// SIMATIC STEP 7 (V5.x) project PLC_MST_WorkingClapans
// CPU: CPU 315-2 PN/DP
// station: P_ADR_BUS
// station: Hardware
// station: SIMATIC 300(2)(1)
// program: S7 Program(5)

SYMBOL_TABLE
"Arrays"	DB 1	DB 1
"Oscilation"	FB 1	FB 1
"S-Walce"	FB 2	FB 2
"GS Bottom&Top Sprusk"	FB 3	FB 3
"Hihgt Preassure Clapan"	FB 4	FB 4
"Service&Work"	FB 5	FB 5
"x0"	I 0.0	BOOL	// кн.Режим работы 1 пресс
"x1"	I 0.1	BOOL	// кн.Режим сервиса 1 пресс
"x2"	I 0.2	BOOL	// 1 Пресс прижать
"x3"	I 0.3	BOOL	// 1 пресс отжать
"x4"	I 0.4	BOOL	// кн.Режим работы 2 пресс работа
"x5"	I 0.5	BOOL	// кн.Режим работы 2 пресс сервис
"x6"	I 0.6	BOOL	// 2 Пресс прижать
"x7"	I 0.7	BOOL	// 2 пресс отжать
"x8"	I 1.0	BOOL	// Кн.Режм работы 3 пресс работа
"x9"	I 1.1	BOOL	// кн.Режим работы 3 пресс сервис
"x10"	I 1.2	BOOL	// 3 Пресс прижать
"x11"	I 1.3	BOOL	// 3 Пресс отжать
"x12"	I 1.4	BOOL	// кн.Осциляци выского давления сетка вкл
"x13"	I 1.5	BOOL	// кн.Осциляция высокого давления 1 пресс
"x14"	I 1.6	BOOL	// кн.Осциляция высокого давления 2 пресс вкл
"x15"	I 1.7	BOOL	// кн.Осциляция выского давления 3 пресс вкл
"x16"	I 2.0	BOOL	// кн.Клапан высокого давления сетка
"x17"	I 2.1	BOOL	// кн.Высокое давление 1 пресс
"x18"	I 2.2	BOOL	// кн. Включить Клапан высокого давления пресс 2
"x19"	I 2.3	BOOL	// кн.Клапан высокого давления 3 пресс
"x20"	I 2.4	BOOL	// кн.Осциляция орошения сукна 1 пресс
"x21"	I 2.5	BOOL	// кн.Осциляция орошения сукна 2 пресс
"x22"	I 2.6	BOOL	// Гидростанция прижима А
"x23"	I 2.7	BOOL	// Гидростанция прижима А пуск
"x24"	I 3.0	BOOL	// Гидростанция прижима В
"x25"	I 3.1	BOOL	// Гидростанция прижима В пуск
"x26"	I 3.2	BOOL	// кн.Гидростанция S-Walce A
"x27"	I 3.3	BOOL	// кн.Гидростанция S-Walce A пуск
"x28"	I 3.4	BOOL	// кн.Гидростанция S-Walce В
"x29"	I 3.5	BOOL	// кн.Гидростанция S-Walce В пуск
"x30"	I 3.6	BOOL	// кн.Вкл Гидростанция спрысков нижняя
"x31"	I 3.7	BOOL	// кн.Выкл Гидростанция спрысков нижняя
"x32"	I 4.0	BOOL	// кн.Вкл Нидростанция спрысков нижняя
"x33"	I 4.1	BOOL	// кн.Выкл Гидростанция спрысков верхняя
"x34"	I 4.2	BOOL	// кн.Стоп 1 пресс
"x35"	I 4.3	BOOL	// кн.Снять 1 пресс
"x36"	I 4.4	BOOL	// кн.Подвести 1 пресс
"x37"	I 4.5	BOOL	// кн.Прижим 1 пресс
"x38"	I 4.6	BOOL	// кн.Стоп 2 пресс
"x39"	I 4.7	BOOL	// кн.Снять 2 пресс
"x40"	I 5.0	BOOL	// кн.Подвести 2 пресс
"x41"	I 5.1	BOOL	// кн.Прижать 2 пресс
"x42"	I 5.2	BOOL	// Замок выкл
"x43"	I 5.3	BOOL	// Замок вкл
"x44"	I 5.4	BOOL	// кн.Стоп 3 пресс
"x45"	I 5.5	BOOL	// кн.Снять 3 пресс
"x46"	I 5.6	BOOL	// кн.Подвести 3 пресс
"x47"	I 5.7	BOOL	// кн.Прижать 3 пресс
"x48"	I 6.0	BOOL	// кн.Облегчть 3 пресс
"x49"	I 6.1	BOOL	// кн.Бомбировка 3 пресс выкл
"x50"	I 6.2	BOOL	// кн.Бомбировка 3 пресс вкл
"x51"	I 6.3	BOOL	// кн.Прижать сеткоповоротный вал
"x52"	I 6.4	BOOL	// кн.Прижим передающий вал 2
"x53"	I 6.5	BOOL	// кн.Прижать передающий вал 3 пресс
"x54"	I 6.6	BOOL	// Замок открыт
"x55"	I 6.7	BOOL	// Замок закрыт
"x56"	I 7.0	BOOL	// Замок открыт
"x57"	I 7.1	BOOL	// Замок закрыт
"x58"	I 7.2	BOOL
"x59"	I 7.3	BOOL
"x60"	I 7.4	BOOL
"x61"	I 7.5	BOOL
"x62"	I 7.6	BOOL
"x63"	I 7.7	BOOL
"x64"	I 8.0	BOOL
"x65"	I 8.1	BOOL
"x66"	I 8.2	BOOL
"x67"	I 8.3	BOOL
"x68"	I 8.4	BOOL
"x69"	I 8.5	BOOL
"x70"	I 8.6	BOOL
"x71"	I 8.7	BOOL
"x72"	I 9.0	BOOL
"x73"	I 9.1	BOOL
"x74"	I 9.2	BOOL
"x75"	I 9.3	BOOL
"x76"	I 9.4	BOOL
"x77"	I 9.5	BOOL
"x78"	I 9.6	BOOL
"x79"	I 9.7	BOOL
"x80"	I 10.0	BOOL
"x81"	I 10.1	BOOL
"x82"	I 10.2	BOOL
"x83"	I 10.3	BOOL
"x84"	I 10.4	BOOL
"x85"	I 10.5	BOOL
"x86"	I 10.6	BOOL
"x87"	I 10.7	BOOL
"x88"	I 11.0	BOOL
"x89"	I 11.1	BOOL
"x90"	I 11.2	BOOL
"x91"	I 11.3	BOOL
"x92"	I 11.4	BOOL
"x93"	I 11.5	BOOL
"x94"	I 11.6	BOOL
"x95"	I 11.7	BOOL
"x96"	I 12.0	BOOL
"x100"	I 12.1	BOOL
"x97"	I 12.2	BOOL
"x101"	I 12.3	BOOL
"x98"	I 12.4	BOOL
"x102"	I 12.5	BOOL
"x99"	I 12.6	BOOL
"x103"	I 12.7	BOOL
"x104"	I 13.0	BOOL
"x108"	I 13.1	BOOL
"x105"	I 13.2	BOOL
"x109"	I 13.3	BOOL
"x106"	I 13.4	BOOL
"x110"	I 13.5	BOOL
"x107"	I 13.6	BOOL
"x111"	I 13.7	BOOL
"x112"	I 14.0	BOOL
"x116"	I 14.1	BOOL
"x113"	I 14.2	BOOL
"x117"	I 14.3	BOOL
"x114"	I 14.4	BOOL
"x118"	I 14.5	BOOL
"x115"	I 14.6	BOOL
"x119"	I 14.7	BOOL
"x120"	I 15.0	BOOL
"x124"	I 15.1	BOOL
"x121"	I 15.2	BOOL
"x125"	I 15.3	BOOL
"x122"	I 15.4	BOOL
"x126"	I 15.5	BOOL
"x123"	I 15.6	BOOL
"x127"	I 15.7	BOOL
"x128"	I 16.0	BOOL
"x132"	I 16.1	BOOL
"x129"	I 16.2	BOOL
"x133"	I 16.3	BOOL
"x130"	I 16.4	BOOL
"x134"	I 16.5	BOOL
"x131"	I 16.6	BOOL
"x135"	I 16.7	BOOL
"x136"	I 17.0	BOOL
"x140"	I 17.1	BOOL
"x137"	I 17.2	BOOL
"x141"	I 17.3	BOOL
"x138"	I 17.4	BOOL
"x142"	I 17.5	BOOL
"x139"	I 17.6	BOOL
"x143"	I 17.7	BOOL
"x144"	I 18.0	BOOL
"x148"	I 18.1	BOOL
"x145"	I 18.2	BOOL
"x149"	I 18.3	BOOL
"x146"	I 18.4	BOOL
"x150"	I 18.5	BOOL
"x147"	I 18.6	BOOL
"x151"	I 18.7	BOOL
"x152"	I 19.0	BOOL
"x156"	I 19.1	BOOL
"x153"	I 19.2	BOOL
"x157"	I 19.3	BOOL
"x154"	I 19.4	BOOL
"x158"	I 19.5	BOOL
"x155"	I 19.6	BOOL
"x159"	I 19.7	BOOL
"x160"	I 20.0	BOOL
"x164"	I 20.1	BOOL
"x161"	I 20.2	BOOL
"x165"	I 20.3	BOOL
"x162"	I 20.4	BOOL
"x166"	I 20.5	BOOL
"x163"	I 20.6	BOOL
"x167"	I 20.7	BOOL
"x168"	I 21.0	BOOL
"x172"	I 21.1	BOOL
"x169"	I 21.2	BOOL
"x173"	I 21.3	BOOL
"x170"	I 21.4	BOOL
"x174"	I 21.5	BOOL
"x171"	I 21.6	BOOL
"x175"	I 21.7	BOOL
"x176"	I 22.0	BOOL
"x180"	I 22.1	BOOL
"x177"	I 22.2	BOOL
"x181"	I 22.3	BOOL
"x178"	I 22.4	BOOL
"x182"	I 22.5	BOOL
"x179"	I 22.6	BOOL
"x183"	I 22.7	BOOL
"x184"	I 23.0	BOOL
"x188"	I 23.1	BOOL
"x185"	I 23.2	BOOL
"x189"	I 23.3	BOOL
"x186"	I 23.4	BOOL
"x190"	I 23.5	BOOL
"x187"	I 23.6	BOOL
"x191"	I 23.7	BOOL
"x192"	I 24.0	BOOL
"x196"	I 24.1	BOOL
"x193"	I 24.2	BOOL
"x197"	I 24.3	BOOL
"x194"	I 24.4	BOOL
"x198"	I 24.5	BOOL
"x195"	I 24.6	BOOL
"x199"	I 24.7	BOOL
"x200"	I 25.0	BOOL
"x204"	I 25.1	BOOL
"x201"	I 25.2	BOOL
"x205"	I 25.3	BOOL
"x202"	I 25.4	BOOL
"x206"	I 25.5	BOOL
"x203"	I 25.6	BOOL
"x207"	I 25.7	BOOL
"x208"	I 26.0	BOOL
"x212"	I 26.1	BOOL
"x209"	I 26.2	BOOL
"x213"	I 26.3	BOOL
"x210"	I 26.4	BOOL
"x214"	I 26.5	BOOL
"x211"	I 26.6	BOOL
"x215"	I 26.7	BOOL
"x216"	I 27.0	BOOL
"x220"	I 27.1	BOOL
"x217"	I 27.2	BOOL
"x221"	I 27.3	BOOL
"x218"	I 27.4	BOOL
"x222"	I 27.5	BOOL
"x219"	I 27.6	BOOL
"x223"	I 27.7	BOOL
"x224"	I 28.0	BOOL
"x228"	I 28.1	BOOL
"x225"	I 28.2	BOOL
"x229"	I 28.3	BOOL
"x226"	I 28.4	BOOL
"x230"	I 28.5	BOOL
"x227"	I 28.6	BOOL	// Проток есть на 3 прессе
"x231"	I 28.7	BOOL
"x232"	I 29.0	BOOL
"x236"	I 29.1	BOOL	// Сигнал с ПРВ,сетка во вращении
"x233"	I 29.2	BOOL
"x237"	I 29.3	BOOL	// Сигнал с ПРВ,работа 3 приводов(1,2 пресс + пикап)
"x234"	I 29.4	BOOL
"x238"	I 29.5	BOOL	// Сигнал с ПРВ,3 пресс в работе
"x235"	I 29.6	BOOL
"x239"	I 29.7	BOOL	// Сигнал работы насос выского давления
"x240"	I 30.0	BOOL
"x244"	I 30.1	BOOL
"x241"	I 30.2	BOOL
"x245"	I 30.3	BOOL
"x242"	I 30.4	BOOL
"x246"	I 30.5	BOOL
"x243"	I 30.6	BOOL
"x247"	I 30.7	BOOL
"x248"	I 31.0	BOOL
"x252"	I 31.1	BOOL
"x249"	I 31.2	BOOL
"x253"	I 31.3	BOOL	// Дискретный датчик температуры ГС 1+3
"x250"	I 31.4	BOOL
"x254"	I 31.5	BOOL	// Дискретный датчик уровня масла ГС 1+3
"x251"	I 31.6	BOOL
"x255"	I 31.7	BOOL
"Delay_2tim"	MW 2	WORD	// Время задержки с панели на включение пресса
"CYCL_EXC"	OB 1	OB 1	// Cycle Execution
"Prog2"	OB 2	OB 2	// S-Walce
"Prog3"	OB 3	OB 3	// Sprusk
"y0"	Q 0.0	BOOL	// Лампа 1 пресс в режиме работы
"y1"	Q 0.1	BOOL	// Лампа пресс 1 в режиме сервис
"y2"	Q 0.2	BOOL	// Лампа 1 пресс прижать
"y3"	Q 0.3	BOOL	// Лампа 1 пресс отжать
"y4"	Q 0.4	BOOL	// Лампа 2 пресс в режиме работы
"y5"	Q 0.5	BOOL	// Лампа 2 пресс в режиме сервиса
"y6"	Q 0.6	BOOL	// Лампа 2 пресс прижать
"y7"	Q 0.7	BOOL	// Лампа 2 пресс отжать
"y8"	Q 1.0	BOOL	// Лампа 3 пресс в режиме работы
"y9"	Q 1.1	BOOL	// Лампа 3 пресс в режиме сервиса
"y10"	Q 1.2	BOOL	// Лампа 3 пресс прижать
"y11"	Q 1.3	BOOL	// Лампа 3 пресс отжать
"y12"	Q 1.4	BOOL	// Лампа выключена осциляция высокого давления сетки
"y13"	Q 1.5	BOOL	// Лампа включена рсциляция высокго давления сетка
"y14"	Q 1.6	BOOL	// Лампа выключена осциляция выского давления 1 пресс
"y15"	Q 1.7	BOOL	// Лампа включена Осциляция выского давления 1 пресс
"y16"	Q 2.0	BOOL	// Лампа выключена осциляция выского давления 2 пресс
"y17"	Q 2.1	BOOL	// Лампа включена осциляция выского давления 2 пресс
"y18"	Q 2.2	BOOL	// Лампа выключена осциляция высокого давления 3 пресс
"y19"	Q 2.3	BOOL	// Лампа включена осциляция высокого давления 3 пресс
"y20"	Q 2.4	BOOL	// Лампа выключен клапан высокого давления сетка
"y21"	Q 2.5	BOOL	// Лампа включен клапан высокого давления сетка
"y22"	Q 2.6	BOOL	// Лампа выключен клапан высокого давления пресс 1
"y23"	Q 2.7	BOOL	// Лампа включен Клапан высокого давления 1 пресс
"y24"	Q 3.0	BOOL	// Лампа выключен клапан высокого давления пресс 2
"y25"	Q 3.1	BOOL	// Лампа включен клапан высокого давления пресс 2
"y26"	Q 3.2	BOOL	// Лампа выключен клапан высокого давления пресс 3
"y27"	Q 3.3	BOOL	// Лампа включен клапан высокого давления пресс 3
"y28"	Q 3.4	BOOL	// Лампа выключена осциляция орошающего спрыска 1 пресс
"y29"	Q 3.5	BOOL	// Лампа включена осциляция орошающего спрыска 1 пресс
"y30"	Q 3.6	BOOL	// Лампа выключена осциляция орошающего спрыска 1 пресс
"y31"	Q 3.7	BOOL	// Лампа включена осциляция орошающего спрыска 2 пресс
"y32"	Q 4.0	BOOL	// Лампа вкл прижим А
"y33"	Q 4.1	BOOL	// Лампа выкл. Гидростанция прижима А&B
"y34"	Q 4.2	BOOL	// Лампа вкл прижим В
"y35"	Q 4.3	BOOL	// Лампа работы гидростанция S-Walke A
"y36"	Q 4.4	BOOL	// Лампа отключен. S-Walke A&B
"y37"	Q 4.5	BOOL	// Лампа работы гидростанция S-Walke B
"y38"	Q 4.6	BOOL	// Лампа выключена ГС спрысков нижняя
"y39"	Q 4.7	BOOL	// Лампа включена ГС спрысков нижняя
"y40"	Q 5.0	BOOL	// Лампа выключена ГС спрысков верхняя
"y41"	Q 5.1	BOOL	// Лампа включена ГС спрысков верхняя
"y42"	Q 5.2	BOOL	// Лампа Стоп 1й прес
"y43"	Q 5.3	BOOL	// Лампа зняти 1й прес
"y44"	Q 5.4	BOOL	// Лампа подвод 1й прес
"y45"	Q 5.5	BOOL	// Лампа прижать 1й прес
"y46"	Q 5.6	BOOL	// Лампа стоп 2й прес
"y47"	Q 5.7	BOOL	// Лампа зняти 2й прес
"y48"	Q 6.0	BOOL	// Лампа подвод 2й прес
"y49"	Q 6.1	BOOL	// Лампа прижати 2й прес
"y50"	Q 6.2	BOOL	// Лампа замок выкл
"y51"	Q 6.3	BOOL	// Лампа замок вкл
"y52"	Q 6.4	BOOL	// Лампа останов 3й прес
"y53"	Q 6.5	BOOL	// Лампа зняти 3й прес
"y54"	Q 6.6	BOOL	// Замок открыт
"y55"	Q 6.7	BOOL	// Лампа прижати 3й прес
"y56"	Q 7.0	BOOL	// Замок открыт
"y57"	Q 7.1	BOOL	// Лампа выключена бомбировка 3 пресс
"y58"	Q 7.2	BOOL	// Лампа включена бомбировка 3 пресс
"y59"	Q 7.3	BOOL	// Бомбировка вкл пресс 3
"y60"	Q 7.4	BOOL	// Клапан замка 1
"y61"	Q 7.5	BOOL	// Клапан замка 2
"y62"	Q 7.6	BOOL
"y63"	Q 7.7	BOOL
"y64"	Q 8.0	BOOL
"y65"	Q 8.1	BOOL
"y66"	Q 8.2	BOOL
"y67"	Q 8.3	BOOL
"y68"	Q 8.4	BOOL
"y69"	Q 8.5	BOOL
"y70"	Q 8.6	BOOL
"y71"	Q 8.7	BOOL
"y72"	Q 9.0	BOOL
"y73"	Q 9.1	BOOL
"y74"	Q 9.2	BOOL
"y75"	Q 9.3	BOOL
"y76"	Q 9.4	BOOL
"y77"	Q 9.5	BOOL
"y78"	Q 9.6	BOOL
"y79"	Q 9.7	BOOL
"y80"	Q 10.0	BOOL
"y81"	Q 10.1	BOOL
"y82"	Q 10.2	BOOL
"y83"	Q 10.3	BOOL
"y84"	Q 10.4	BOOL
"y85"	Q 10.5	BOOL
"y86"	Q 10.6	BOOL
"y87"	Q 10.7	BOOL
"y88"	Q 11.0	BOOL
"y89"	Q 11.1	BOOL
"y90"	Q 11.2	BOOL
"y91"	Q 11.3	BOOL
"y92"	Q 11.4	BOOL
"y93"	Q 11.5	BOOL
"y94"	Q 11.6	BOOL
"y95"	Q 11.7	BOOL
"y96"	Q 12.0	BOOL
"y100"	Q 12.1	BOOL
"y97"	Q 12.2	BOOL
"y101"	Q 12.3	BOOL
"y98"	Q 12.4	BOOL
"y102"	Q 12.5	BOOL
"y99"	Q 12.6	BOOL
"y103"	Q 12.7	BOOL	// Гидростанция S-Walce A
"y104"	Q 13.0	BOOL	// Гидростанция S-Walce В
"y108"	Q 13.1	BOOL
"y105"	Q 13.2	BOOL
"y109"	Q 13.3	BOOL
"y106"	Q 13.4	BOOL
"y110"	Q 13.5	BOOL
"y107"	Q 13.6	BOOL
"y111"	Q 13.7	BOOL	// Гидростанция спрысков верхняя
"y112"	Q 14.0	BOOL	// Гидростанция прижима А
"y116"	Q 14.1	BOOL
"y113"	Q 14.2	BOOL	// Гидростанция спырсков нижняя
"y117"	Q 14.3	BOOL
"y114"	Q 14.4	BOOL	// Гидростанция прижима В
"y118"	Q 14.5	BOOL
"y115"	Q 14.6	BOOL
"y119"	Q 14.7	BOOL
"y120"	Q 15.0	BOOL
"y124"	Q 15.1	BOOL	// Клапан ГС спрысков верхний
"y121"	Q 15.2	BOOL
"y125"	Q 15.3	BOOL
"y122"	Q 15.4	BOOL
"y126"	Q 15.5	BOOL	// Клапан высокого давления пресс 1
"y123"	Q 15.6	BOOL
"y127"	Q 15.7	BOOL	// Клапан высокго давления пресс 2
"y128"	Q 16.0	BOOL	// Клапан высокого давления пресс 3
"y132"	Q 16.1	BOOL
"y129"	Q 16.2	BOOL	// Клапан высокого давления сетка
"y133"	Q 16.3	BOOL	// WE3 2 PRESS
"y130"	Q 16.4	BOOL	// Сигнал на ПРВ, Дозвіл работы 1,2 пресса+пикап
"y134"	Q 16.5	BOOL	// WE2 2 PRESS
"y131"	Q 16.6	BOOL	// Сигнал на ПРВ,Запрет включения 3 пресса
"y135"	Q 16.7	BOOL	// WE1.1 2 PRESS
"y136"	Q 17.0	BOOL	// WE 1.2 2PRESS
"y140"	Q 17.1	BOOL
"y137"	Q 17.2	BOOL	// 2 пресс отжать
"y141"	Q 17.3	BOOL	// Прижим передающий вал 2 пресс
"y138"	Q 17.4	BOOL	// 2 пресс прижать
"y142"	Q 17.5	BOOL	// Отжать передающий вал 3 пресс
"y139"	Q 17.6	BOOL
"y143"	Q 17.7	BOOL	// Прижать передающий вал 3 пресс
"y144"	Q 18.0	BOOL	// Прижать сеткоповоротный вал
"y148"	Q 18.1	BOOL	// WE5.1 3 PRESS
"y145"	Q 18.2	BOOL	// WE3 1 PRESS
"y149"	Q 18.3	BOOL	// WE5.2 3 PRESS
"y146"	Q 18.4	BOOL	// WE2.1 1 PRESS
"y150"	Q 18.5	BOOL	// WE4.1 3 PRESS
"y147"	Q 18.6	BOOL	// WE2.2 1 PRESS
"y151"	Q 18.7	BOOL	// WE 4.2 3 PRESS
"y152"	Q 19.0	BOOL	// WE6 3 PRESS
"y156"	Q 19.1	BOOL	// 1 пресс прижать
"y153"	Q 19.2	BOOL	// 1 пресс прижать WE4
"y157"	Q 19.3	BOOL	// 1 пресс отжать WE4
"y154"	Q 19.4	BOOL	// 1 пресс прижать WE4 A
"y158"	Q 19.5	BOOL
"y155"	Q 19.6	BOOL	// 1 пресс отжать WE4 A
"y159"	Q 19.7	BOOL
"y160"	Q 20.0	BOOL	// 3 пресс прижать
"y164"	Q 20.1	BOOL	// Клапан осциляции выского давления 1 пресс
"y161"	Q 20.2	BOOL	// 3 пресс отжать
"y165"	Q 20.3	BOOL
"y162"	Q 20.4	BOOL	// Клапан осциляции высокого давления сетки
"y166"	Q 20.5	BOOL	// Клапан осциляции выского давления 2 пресс
"y163"	Q 20.6	BOOL	// Клапан осциляции выского давления 3 пресс
"y167"	Q 20.7	BOOL
"t0"	T 0	TIMER	// Таймер прерывания 1с
"t1"	T 1	TIMER	// Таймер прерывания 1с
"t2"	T 2	TIMER	// Задержка на разрешение включения пресса
"t3"	T 3	TIMER	// Задержка на разрешение включения пресса
"VAT_1"	VAT 1	
END_SYMBOL_TABLE

FUNCTION_BLOCK "Oscilation"	// FB 1
VERSION : 0.1
VAR_TEMP
  DatArray : ARRAY  [0 .. 5 ] OF INT ;
END_VAR
BEGIN
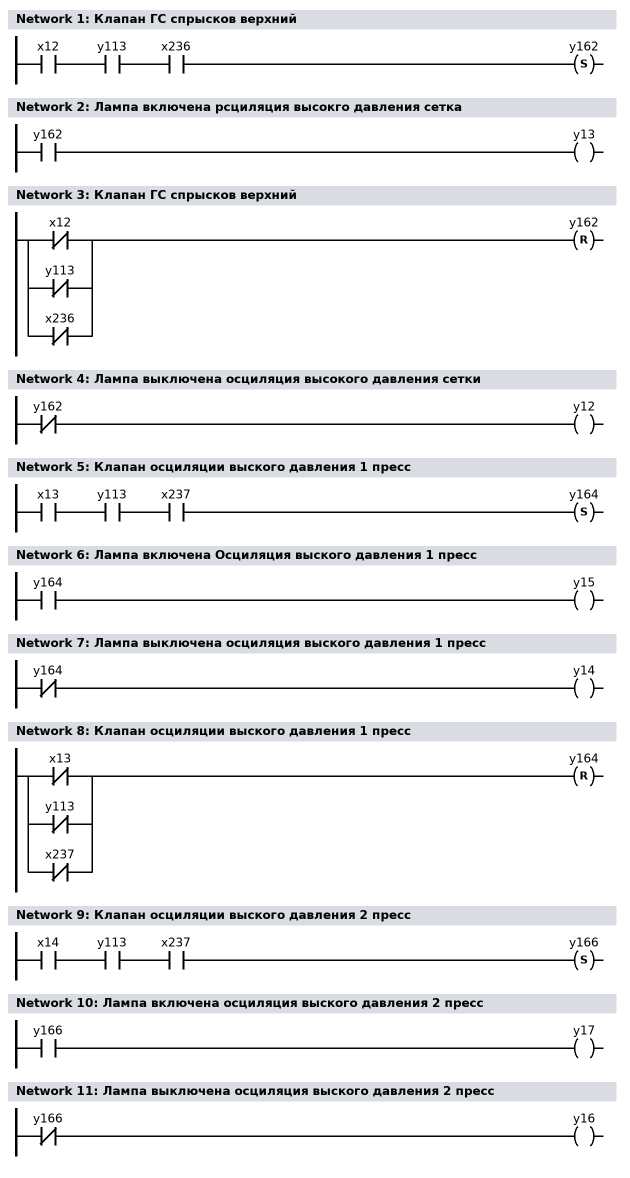
NETWORK
TITLE = Клапан ГС спрысков верхний
      A     "x12";
      A     "y113";
      A     "x236";
      S     "y162";
NETWORK
TITLE = Лампа включена рсциляция высокго давления сетка
      A     "y162";
      =     "y13";
NETWORK
TITLE = Клапан ГС спрысков верхний
      ON    "x12";
      ON    "y113";
      ON    "x236";
      R     "y162";
NETWORK
TITLE = Лампа выключена осциляция высокого давления сетки
      AN    "y162";
      =     "y12";
NETWORK
TITLE = Клапан осциляции выского давления 1 пресс
      A     "x13";
      A     "y113";
      A     "x237";
      S     "y164";
NETWORK
TITLE = Лампа включена Осциляция выского давления 1 пресс
      A     "y164";
      =     "y15";
NETWORK
TITLE = Лампа выключена осциляция выского давления 1 пресс
      AN    "y164";
      =     "y14";
NETWORK
TITLE = Клапан осциляции выского давления 1 пресс
      ON    "x13";
      ON    "y113";
      ON    "x237";
      R     "y164";
NETWORK
TITLE = Клапан осциляции выского давления 2 пресс
      A     "x14";
      A     "y113";
      A     "x237";
      S     "y166";
NETWORK
TITLE = Лампа включена осциляция выского давления 2 пресс
      A     "y166";
      =     "y17";
NETWORK
TITLE = Лампа выключена осциляция выского давления 2 пресс
      AN    "y166";
      =     "y16";
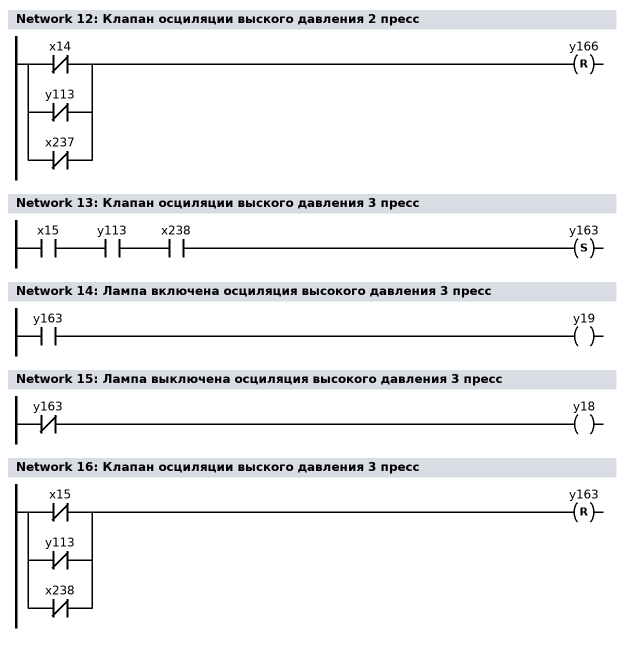
NETWORK
TITLE = Клапан осциляции выского давления 2 пресс
      ON    "x14";
      ON    "y113";
      ON    "x237";
      R     "y166";
NETWORK
TITLE = Клапан осциляции выского давления 3 пресс
      A     "x15";
      A     "y113";
      A     "x238";
      S     "y163";
NETWORK
TITLE = Лампа включена осциляция высокого давления 3 пресс
      A     "y163";
      =     "y19";
NETWORK
TITLE = Лампа выключена осциляция высокого давления 3 пресс
      AN    "y163";
      =     "y18";
NETWORK
TITLE = Клапан осциляции выского давления 3 пресс
      ON    "x15";
      ON    "y113";
      ON    "x238";
      R     "y163";
END_FUNCTION_BLOCK

FUNCTION_BLOCK "S-Walce"	// FB 2
VERSION : 0.1
BEGIN
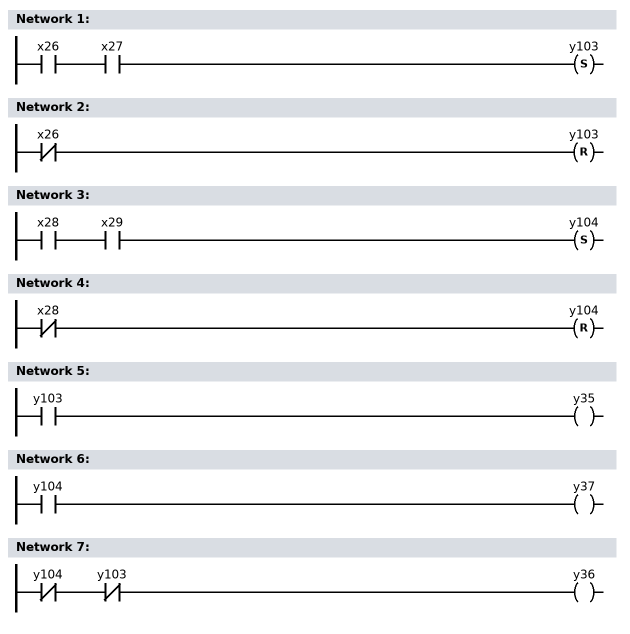
NETWORK
TITLE =
      A     "x26";
      A     "x27";
      S     "y103";
NETWORK
TITLE =
      AN    "x26";
      R     "y103";
NETWORK
TITLE =
      A     "x28";
      A     "x29";
      S     "y104";
NETWORK
TITLE =
      AN    "x28";
      R     "y104";
NETWORK
TITLE =
      A     "y103";
      =     "y35";
NETWORK
TITLE =
      A     "y104";
      =     "y37";
NETWORK
TITLE =
      AN    "y104";
      AN    "y103";
      =     "y36";
END_FUNCTION_BLOCK

FUNCTION_BLOCK "GS Bottom&Top Sprusk"	// FB 3
VERSION : 0.1
VAR_TEMP
  m0 : BOOL ;	//Аварийный сигнал с ГС 1+3
END_VAR
BEGIN
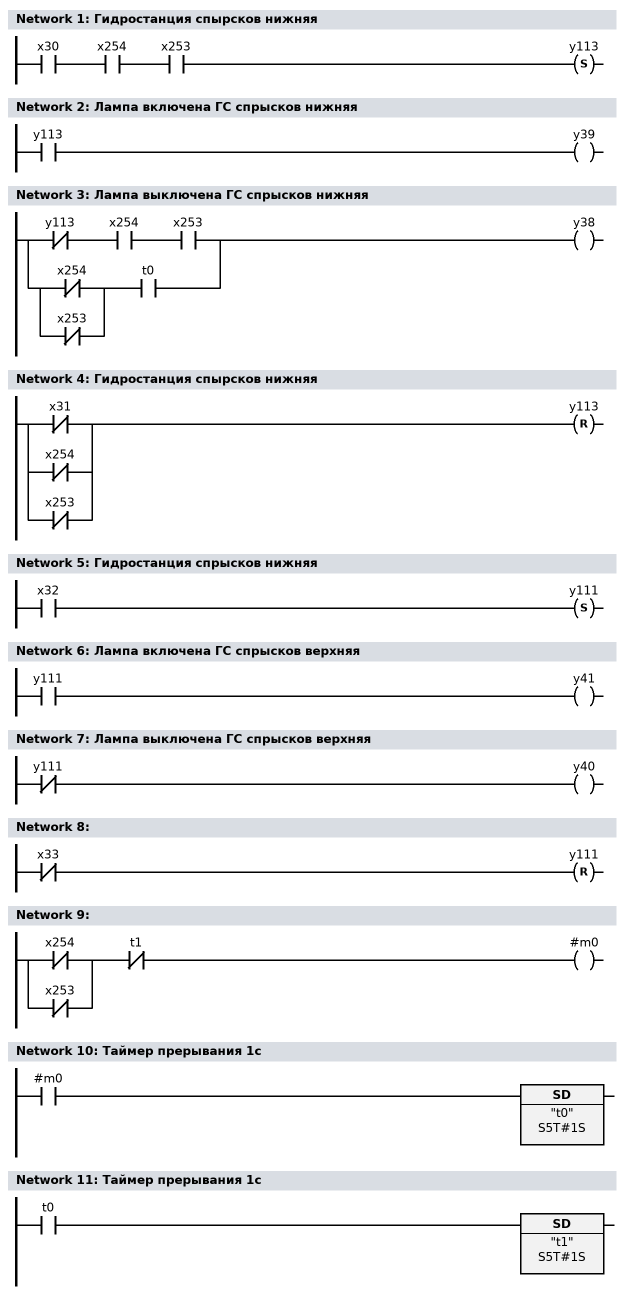
NETWORK
TITLE = Гидростанция спырсков нижняя
      A     "x30";
      A     "x254";
      A     "x253";
      S     "y113";
NETWORK
TITLE = Лампа включена ГС спрысков нижняя
      A     "y113";
      =     "y39";
NETWORK
TITLE = Лампа выключена ГС спрысков нижняя
      AN    "y113";
      A     "x254";
      A     "x253";
      O;
      A(;
      ON    "x254";
      ON    "x253";
      );
      A     "t0";
      =     "y38";
NETWORK
TITLE = Гидростанция спырсков нижняя
      ON    "x31";
      ON    "x254";
      ON    "x253";
      R     "y113";
NETWORK
TITLE = Гидростанция спрысков нижняя
      A     "x32";
      S     "y111";
NETWORK
TITLE = Лампа включена ГС спрысков верхняя
      A     "y111";
      =     "y41";
NETWORK
TITLE = Лампа выключена ГС спрысков верхняя
      AN    "y111";
      =     "y40";
NETWORK
TITLE =
      AN    "x33";
      R     "y111";
NETWORK
TITLE =
//<force open>
      A(;
      ON    "x254";
      ON    "x253";
      );
      AN    "t1";
      =     #m0;
NETWORK
TITLE = Таймер прерывания 1с
      A     #m0;
      L     S5T#1S;
      SD    "t0";
NETWORK
TITLE = Таймер прерывания 1с
      A     "t0";
      L     S5T#1S;
      SD    "t1";
END_FUNCTION_BLOCK

FUNCTION_BLOCK "Hihgt Preassure Clapan"	// FB 4
TITLE = Hight Pressure Klapan
VERSION : 0.1
BEGIN
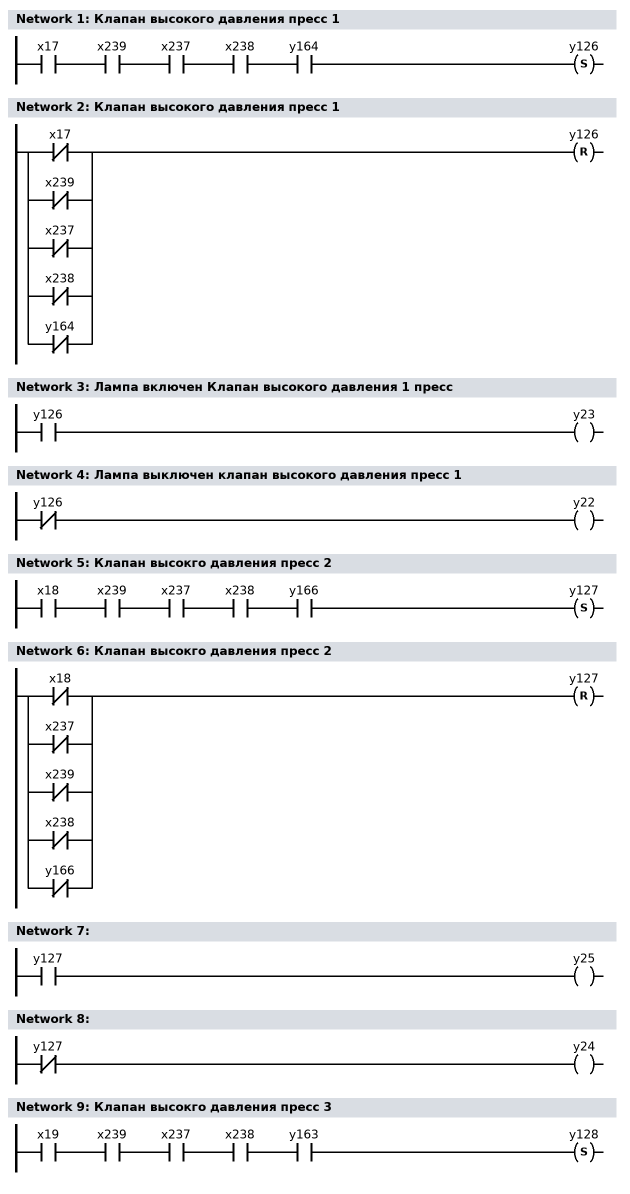
NETWORK
TITLE = Клапан высокого давления пресс 1
      A     "x17";
      A     "x239";
      A     "x237";
      A     "x238";
      A     "y164";
      S     "y126";
NETWORK
TITLE = Клапан высокого давления пресс 1
      ON    "x17";
      ON    "x239";
      ON    "x237";
      ON    "x238";
      ON    "y164";
      R     "y126";
NETWORK
TITLE = Лампа включен Клапан высокого давления 1 пресс
      A     "y126";
      =     "y23";
NETWORK
TITLE = Лампа выключен клапан высокого давления пресс 1
      AN    "y126";
      =     "y22";
NETWORK
TITLE = Клапан высокго давления пресс 2
      A     "x18";
      A     "x239";
      A     "x237";
      A     "x238";
      A     "y166";
      S     "y127";
NETWORK
TITLE = Клапан высокго давления пресс 2
      ON    "x18";
      ON    "x237";
      ON    "x239";
      ON    "x238";
      ON    "y166";
      R     "y127";
NETWORK
TITLE =
      A     "y127";
      =     "y25";
NETWORK
TITLE =
      AN    "y127";
      =     "y24";
NETWORK
TITLE = Клапан высокго давления пресс 3
      A     "x19";
      A     "x239";
      A     "x237";
      A     "x238";
      A     "y163";
      S     "y128";
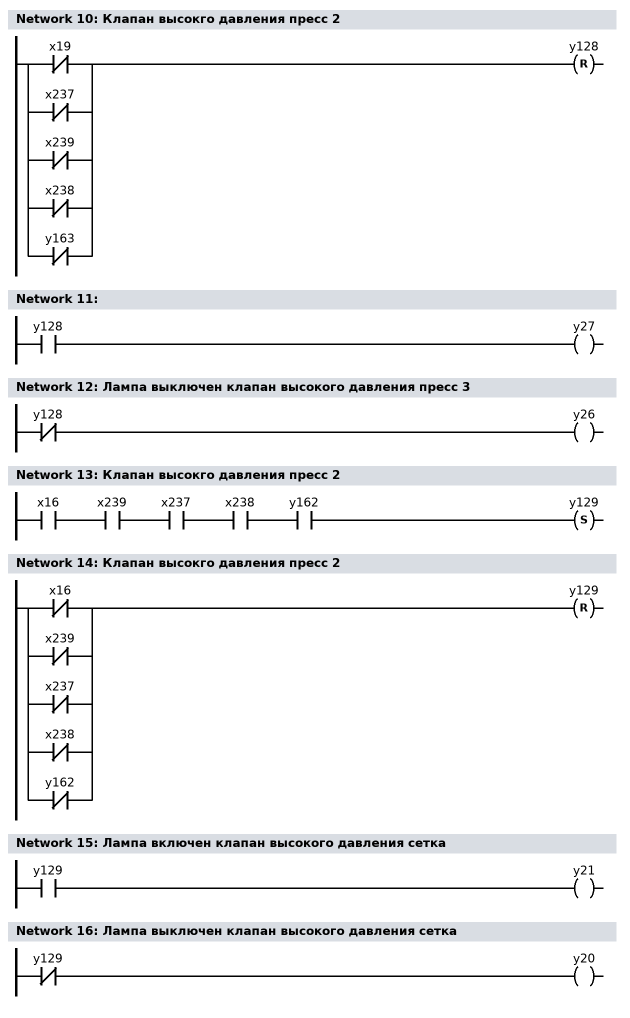
NETWORK
TITLE = Клапан высокго давления пресс 2
      ON    "x19";
      ON    "x237";
      ON    "x239";
      ON    "x238";
      ON    "y163";
      R     "y128";
NETWORK
TITLE =
      A     "y128";
      =     "y27";
NETWORK
TITLE = Лампа выключен клапан высокого давления пресс 3
      AN    "y128";
      =     "y26";
NETWORK
TITLE = Клапан высокго давления пресс 2
      A     "x16";
      A     "x239";
      A     "x237";
      A     "x238";
      A     "y162";
      S     "y129";
NETWORK
TITLE = Клапан высокго давления пресс 2
      ON    "x16";
      ON    "x239";
      ON    "x237";
      ON    "x238";
      ON    "y162";
      R     "y129";
NETWORK
TITLE = Лампа включен клапан высокого давления сетка
      A     "y129";
      =     "y21";
NETWORK
TITLE = Лампа выключен клапан высокого давления сетка
      AN    "y129";
      =     "y20";
END_FUNCTION_BLOCK

FUNCTION_BLOCK "Service&Work"	// FB 5
//SELECT MODE
//
VERSION : 0.1
VAR_TEMP
  ServiceSelect1Press : BOOL ;	//1 пресс в режиме сервиса
  ServiceSelect2Press : BOOL ;	// 2 пресс в режиме сервиса
  ServiceSelect3Press : BOOL ;	//3 пресс в режиме сервиса
  WorkSelect1Press : BOOL ;	//1 Пресс в режиме работы
  WorkSelect2Press : BOOL ;	//2 пресс в режиме работы
  WorkSelect3Press : BOOL ;	//3 пресс в режиме работы
  Dozvil_Privod_1_2_Press : BOOL ;
  Dozvil_Privod_3_Press : BOOL ;
  Kn_Podvod_1_Press_najata : BOOL ;
  Kn_Podvod_2_Press_najata : BOOL ;
  Kn_Podvod_3_Press_najata : BOOL ;
END_VAR
BEGIN
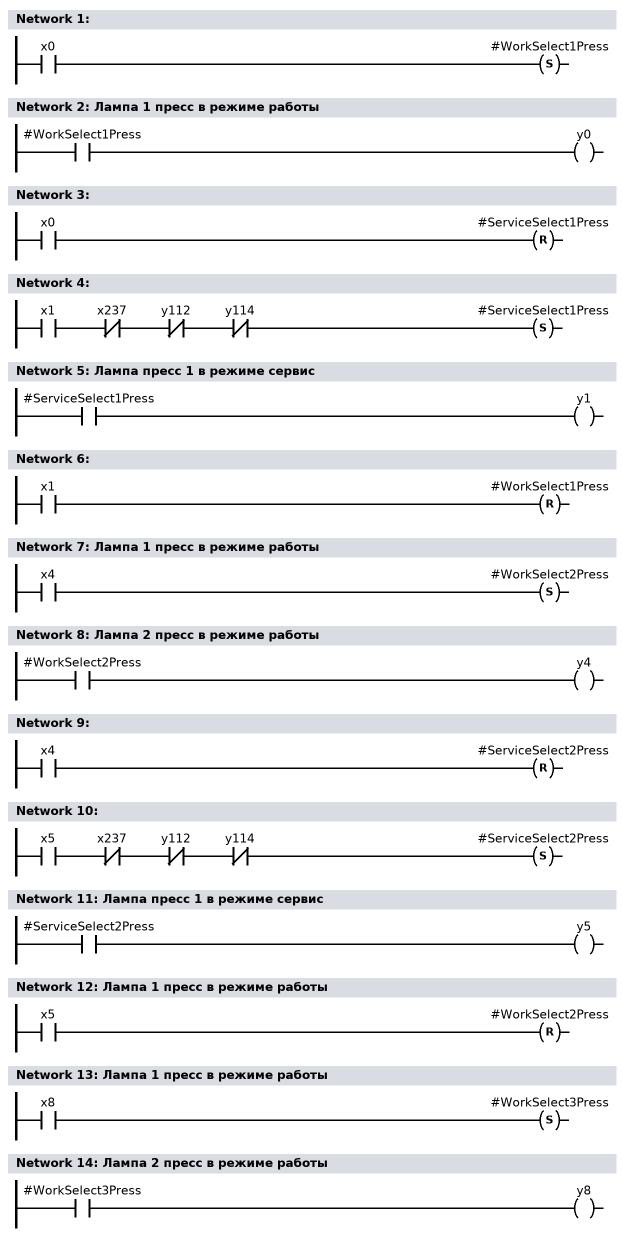
NETWORK
TITLE =
      A     "x0";
      S     #WorkSelect1Press;
NETWORK
TITLE = Лампа 1 пресс в режиме работы
      A     #WorkSelect1Press;
      =     "y0";
NETWORK
TITLE =
      A     "x0";
      R     #ServiceSelect1Press;
NETWORK
TITLE =
      A     "x1";
      AN    "x237";
      AN    "y112";
      AN    "y114";
      S     #ServiceSelect1Press;
NETWORK
TITLE = Лампа пресс 1 в режиме сервис
      A     #ServiceSelect1Press;
      =     "y1";
NETWORK
TITLE =
      A     "x1";
      R     #WorkSelect1Press;
NETWORK
TITLE = Лампа 1 пресс в режиме работы
      A     "x4";
      S     #WorkSelect2Press;
NETWORK
TITLE = Лампа 2 пресс в режиме работы
      A     #WorkSelect2Press;
      =     "y4";
NETWORK
TITLE =
      A     "x4";
      R     #ServiceSelect2Press;
NETWORK
TITLE =
      A     "x5";
      AN    "x237";
      AN    "y112";
      AN    "y114";
      S     #ServiceSelect2Press;
NETWORK
TITLE = Лампа пресс 1 в режиме сервис
      A     #ServiceSelect2Press;
      =     "y5";
NETWORK
TITLE = Лампа 1 пресс в режиме работы
      A     "x5";
      R     #WorkSelect2Press;
NETWORK
TITLE = Лампа 1 пресс в режиме работы
      A     "x8";
      S     #WorkSelect3Press;
NETWORK
TITLE = Лампа 2 пресс в режиме работы
      A     #WorkSelect3Press;
      =     "y8";
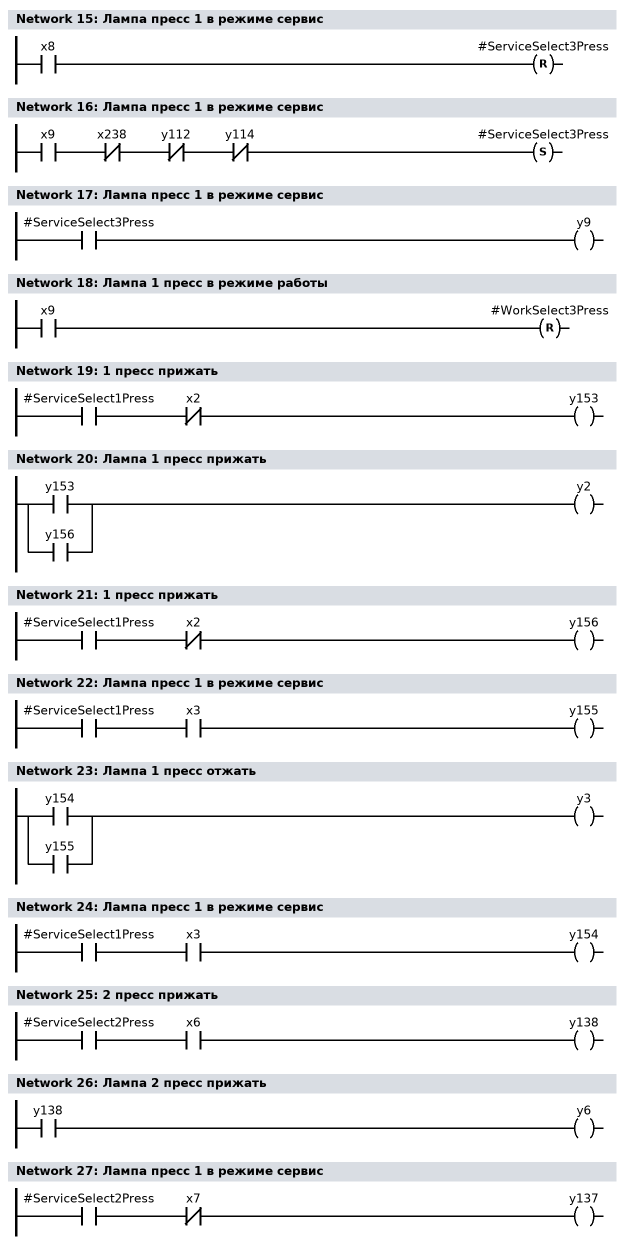
NETWORK
TITLE = Лампа пресс 1 в режиме сервис
      A     "x8";
      R     #ServiceSelect3Press;
NETWORK
TITLE = Лампа пресс 1 в режиме сервис
      A     "x9";
      AN    "x238";
      AN    "y112";
      AN    "y114";
      S     #ServiceSelect3Press;
NETWORK
TITLE = Лампа пресс 1 в режиме сервис
      A     #ServiceSelect3Press;
      =     "y9";
NETWORK
TITLE = Лампа 1 пресс в режиме работы
      A     "x9";
      R     #WorkSelect3Press;
NETWORK
TITLE = 1 пресс прижать
//SERVICE MODE
//
      A     #ServiceSelect1Press;
      AN    "x2";
      =     "y153";
NETWORK
TITLE = Лампа 1 пресс прижать
      O     "y153";
      O     "y156";
      =     "y2";
NETWORK
TITLE = 1 пресс прижать
      A     #ServiceSelect1Press;
      AN    "x2";
      =     "y156";
NETWORK
TITLE = Лампа пресс 1 в режиме сервис
      A     #ServiceSelect1Press;
      A     "x3";
      =     "y155";
NETWORK
TITLE = Лампа 1 пресс отжать
      O     "y154";
      O     "y155";
      =     "y3";
NETWORK
TITLE = Лампа пресс 1 в режиме сервис
      A     #ServiceSelect1Press;
      A     "x3";
      =     "y154";
NETWORK
TITLE = 2 пресс прижать
      A     #ServiceSelect2Press;
      A     "x6";
      =     "y138";
NETWORK
TITLE = Лампа 2 пресс прижать
      A     "y138";
      =     "y6";
NETWORK
TITLE = Лампа пресс 1 в режиме сервис
      A     #ServiceSelect2Press;
      AN    "x7";
      =     "y137";
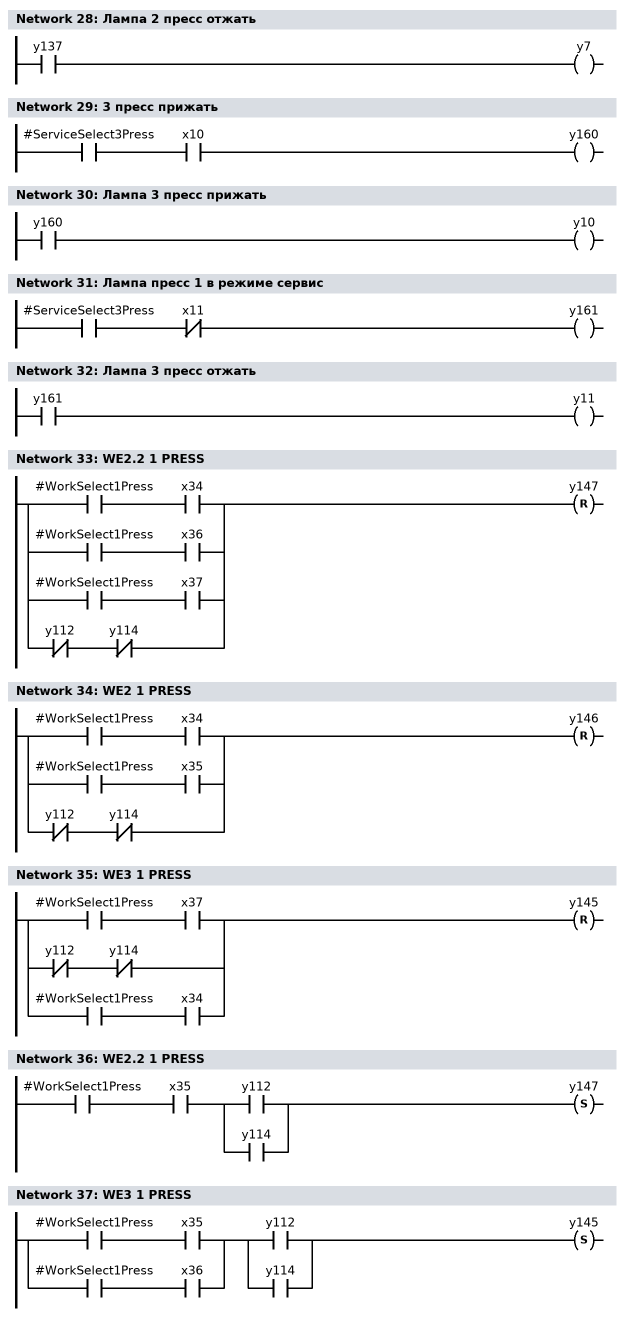
NETWORK
TITLE = Лампа 2 пресс отжать
      A     "y137";
      =     "y7";
NETWORK
TITLE = 3 пресс прижать
      A     #ServiceSelect3Press;
      A     "x10";
      =     "y160";
NETWORK
TITLE = Лампа 3 пресс прижать
      A     "y160";
      =     "y10";
NETWORK
TITLE = Лампа пресс 1 в режиме сервис
      A     #ServiceSelect3Press;
      AN    "x11";
      =     "y161";
NETWORK
TITLE = Лампа 3 пресс отжать
      A     "y161";
      =     "y11";
NETWORK
TITLE = WE2.2 1 PRESS
//WORK MODE
//
      A     #WorkSelect1Press;
      A     "x34";
      O;
      A     #WorkSelect1Press;
      A     "x36";
      O;
      A     #WorkSelect1Press;
      A     "x37";
      O;
      AN    "y112";
      AN    "y114";
      R     "y147";
NETWORK
TITLE = WE2 1 PRESS
      A     #WorkSelect1Press;
      A     "x34";
      O;
      A     #WorkSelect1Press;
      A     "x35";
      O;
      AN    "y112";
      AN    "y114";
      R     "y146";
NETWORK
TITLE = WE3 1 PRESS
      A     #WorkSelect1Press;
      A     "x37";
      O;
      AN    "y112";
      AN    "y114";
      O;
      A     #WorkSelect1Press;
      A     "x34";
      R     "y145";
NETWORK
TITLE = WE2.2 1 PRESS
      A     #WorkSelect1Press;
      A     "x35";
      A(;
      O     "y112";
      O     "y114";
      );
      S     "y147";
NETWORK
TITLE = WE3 1 PRESS
      A(;
      A     #WorkSelect1Press;
      A     "x35";
      O;
      A     #WorkSelect1Press;
      A     "x36";
      );
      A(;
      O     "y112";
      O     "y114";
      );
      S     "y145";
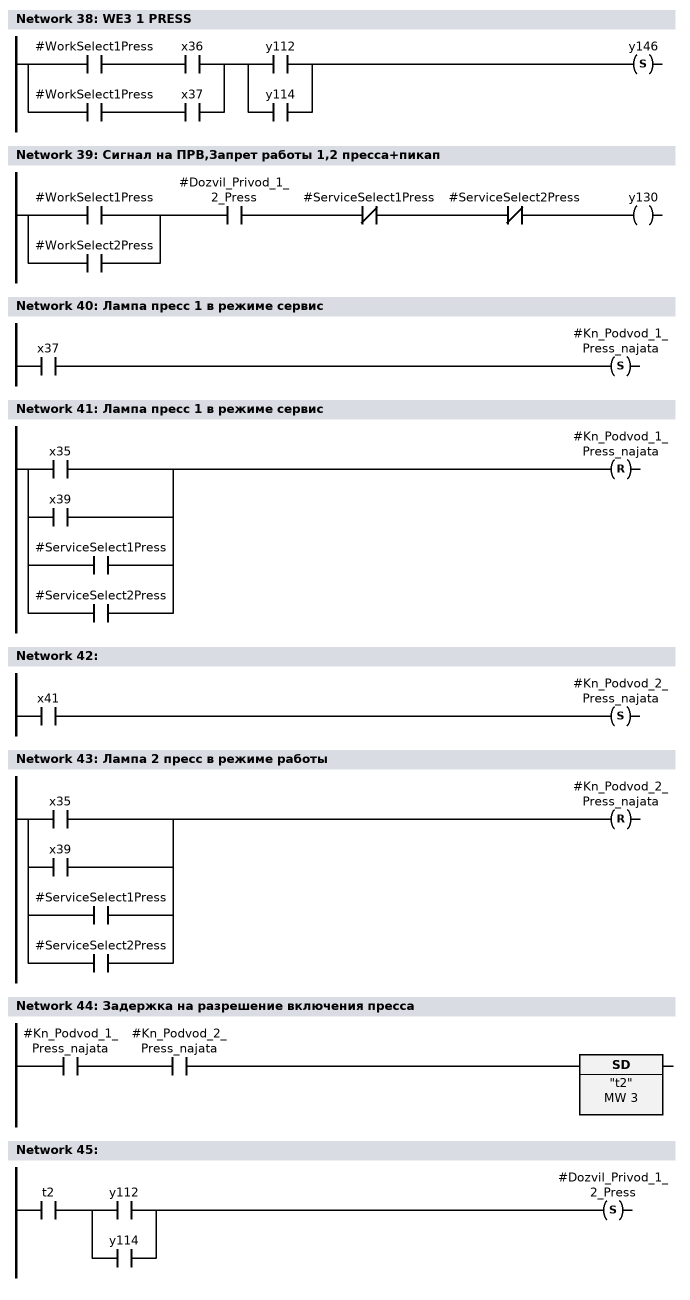
NETWORK
TITLE = WE3 1 PRESS
      A(;
      A     #WorkSelect1Press;
      A     "x36";
      O;
      A     #WorkSelect1Press;
      A     "x37";
      );
      A(;
      O     "y112";
      O     "y114";
      );
      S     "y146";
NETWORK
TITLE = Сигнал на ПРВ,Запрет работы 1,2 пресса+пикап
//Safety
//
      A(;
      O     #WorkSelect1Press;
      O     #WorkSelect2Press;
      );
      A     #Dozvil_Privod_1_2_Press;
      AN    #ServiceSelect1Press;
      AN    #ServiceSelect2Press;
      =     "y130";
NETWORK
TITLE = Лампа пресс 1 в режиме сервис
      A     "x37";
      S     #Kn_Podvod_1_Press_najata;
NETWORK
TITLE = Лампа пресс 1 в режиме сервис
      O     "x35";
      O     "x39";
      O     #ServiceSelect1Press;
      O     #ServiceSelect2Press;
      R     #Kn_Podvod_1_Press_najata;
NETWORK
TITLE =
      A     "x41";
      S     #Kn_Podvod_2_Press_najata;
NETWORK
TITLE = Лампа 2 пресс в режиме работы
      O     "x35";
      O     "x39";
      O     #ServiceSelect1Press;
      O     #ServiceSelect2Press;
      R     #Kn_Podvod_2_Press_najata;
NETWORK
TITLE = Задержка на разрешение включения пресса
      A     #Kn_Podvod_1_Press_najata;
      A     #Kn_Podvod_2_Press_najata;
      L     MW 3;
      SD    "t2";
NETWORK
TITLE =
      A     "t2";
      A(;
      O     "y112";
      O     "y114";
      );
      S     #Dozvil_Privod_1_2_Press;
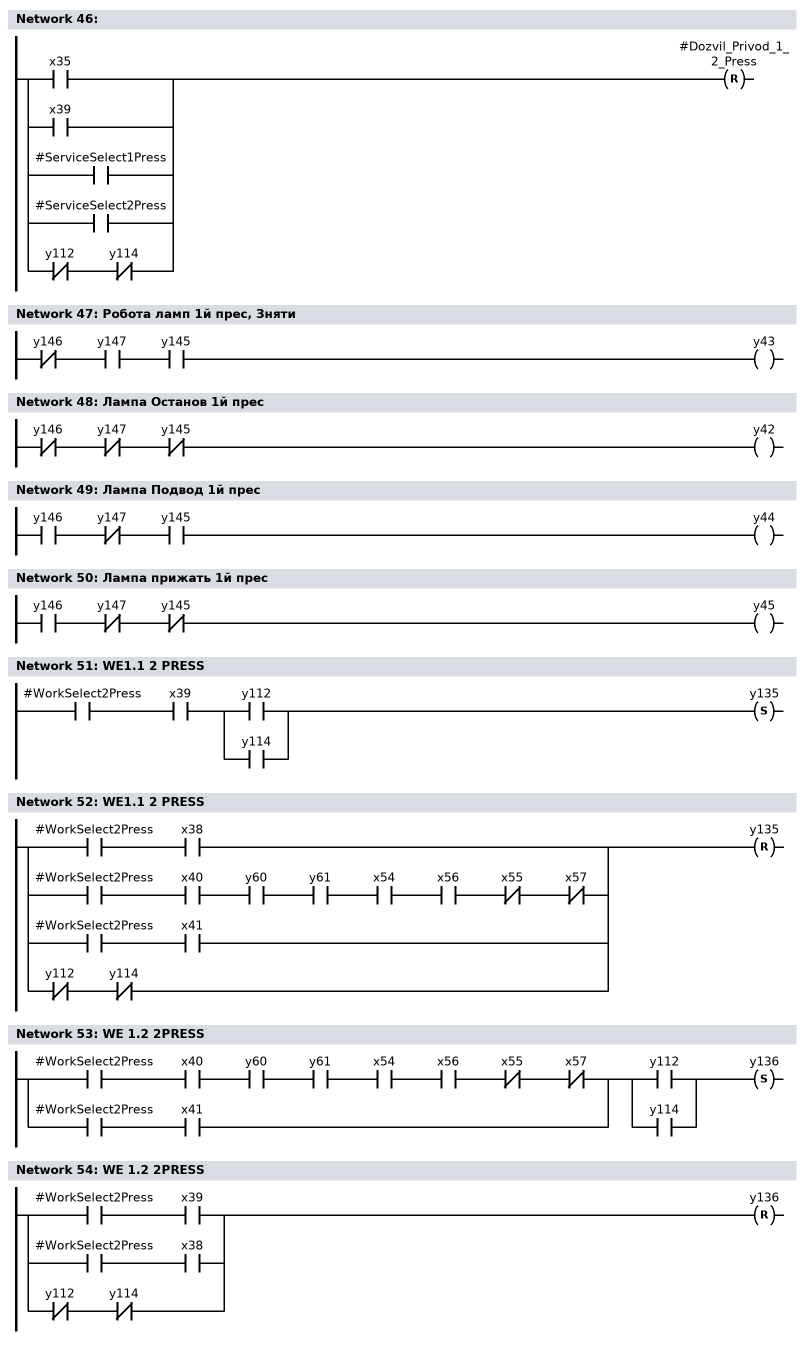
NETWORK
TITLE =
      O     "x35";
      O     "x39";
      O     #ServiceSelect1Press;
      O     #ServiceSelect2Press;
      O;
      AN    "y112";
      AN    "y114";
      R     #Dozvil_Privod_1_2_Press;
NETWORK
TITLE = Робота ламп 1й прес, Зняти
      AN    "y146";
      A     "y147";
      A     "y145";
      =     "y43";
NETWORK
TITLE = Лампа Останов 1й прес
      AN    "y146";
      AN    "y147";
      AN    "y145";
      =     "y42";
NETWORK
TITLE = Лампа Подвод 1й прес
      A     "y146";
      AN    "y147";
      A     "y145";
      =     "y44";
NETWORK
TITLE = Лампа прижать 1й прес
      A     "y146";
      AN    "y147";
      AN    "y145";
      =     "y45";
NETWORK
TITLE = WE1.1 2 PRESS
//WORK SELECTION 2 PRESS
      A     #WorkSelect2Press;
      A     "x39";
      A(;
      O     "y112";
      O     "y114";
      );
      S     "y135";
NETWORK
TITLE = WE1.1 2 PRESS
      A     #WorkSelect2Press;
      A     "x38";
      O;
      A     #WorkSelect2Press;
      A     "x40";
      A     "y60";
      A     "y61";
      A     "x54";
      A     "x56";
      AN    "x55";
      AN    "x57";
      O;
      A     #WorkSelect2Press;
      A     "x41";
      O;
      AN    "y112";
      AN    "y114";
      R     "y135";
NETWORK
TITLE = WE 1.2 2PRESS
      A(;
      A     #WorkSelect2Press;
      A     "x40";
      A     "y60";
      A     "y61";
      A     "x54";
      A     "x56";
      AN    "x55";
      AN    "x57";
      O;
      A     #WorkSelect2Press;
      A     "x41";
      );
      A(;
      O     "y112";
      O     "y114";
      );
      S     "y136";
NETWORK
TITLE = WE 1.2 2PRESS
      A     #WorkSelect2Press;
      A     "x39";
      O;
      A     #WorkSelect2Press;
      A     "x38";
      O;
      AN    "y112";
      AN    "y114";
      R     "y136";
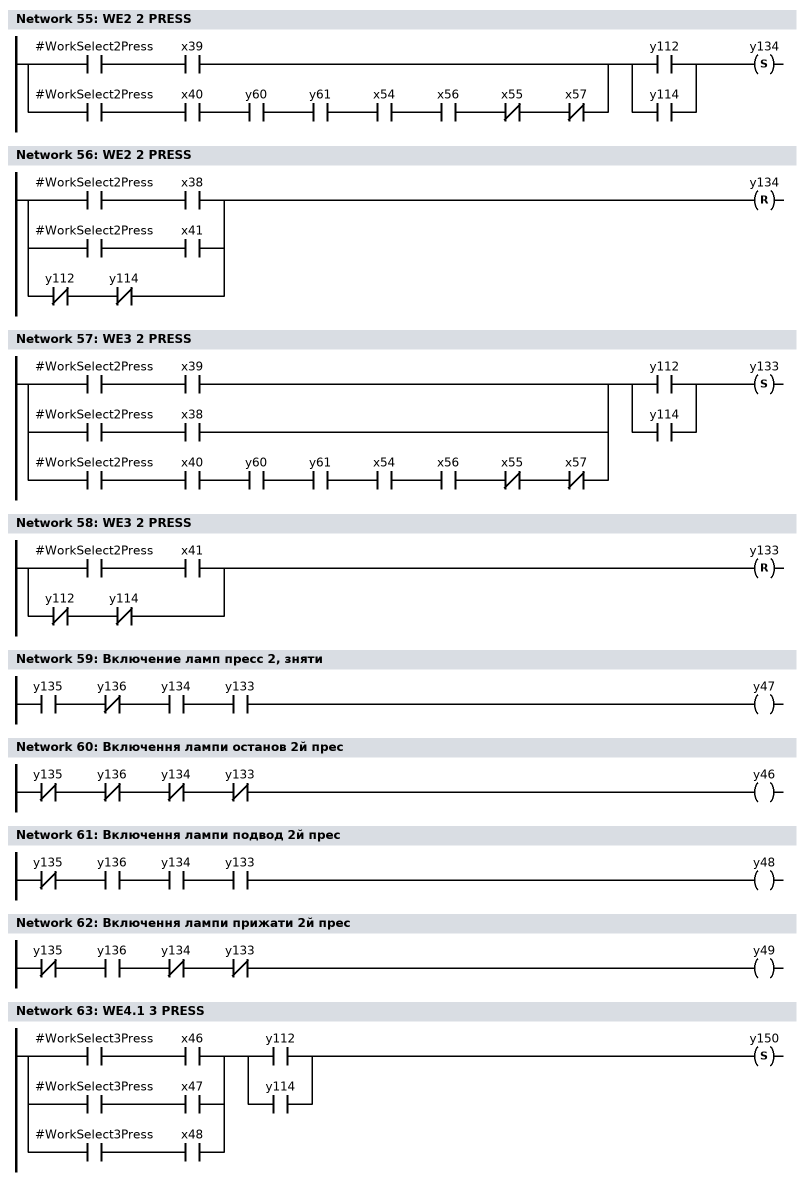
NETWORK
TITLE = WE2 2 PRESS
      A(;
      A     #WorkSelect2Press;
      A     "x39";
      O;
      A     #WorkSelect2Press;
      A     "x40";
      A     "y60";
      A     "y61";
      A     "x54";
      A     "x56";
      AN    "x55";
      AN    "x57";
      );
      A(;
      O     "y112";
      O     "y114";
      );
      S     "y134";
NETWORK
TITLE = WE2 2 PRESS
      A     #WorkSelect2Press;
      A     "x38";
      O;
      A     #WorkSelect2Press;
      A     "x41";
      O;
      AN    "y112";
      AN    "y114";
      R     "y134";
NETWORK
TITLE = WE3 2 PRESS
      A(;
      A     #WorkSelect2Press;
      A     "x39";
      O;
      A     #WorkSelect2Press;
      A     "x38";
      O;
      A     #WorkSelect2Press;
      A     "x40";
      A     "y60";
      A     "y61";
      A     "x54";
      A     "x56";
      AN    "x55";
      AN    "x57";
      );
      A(;
      O     "y112";
      O     "y114";
      );
      S     "y133";
NETWORK
TITLE = WE3 2 PRESS
      A     #WorkSelect2Press;
      A     "x41";
      O;
      AN    "y112";
      AN    "y114";
      R     "y133";
NETWORK
TITLE = Включение ламп пресс 2, зняти 
      A     "y135";
      AN    "y136";
      A     "y134";
      A     "y133";
      =     "y47";
NETWORK
TITLE = Включення лампи останов 2й прес
      AN    "y135";
      AN    "y136";
      AN    "y134";
      AN    "y133";
      =     "y46";
NETWORK
TITLE = Включення лампи подвод 2й прес
      AN    "y135";
      A     "y136";
      A     "y134";
      A     "y133";
      =     "y48";
NETWORK
TITLE = Включення лампи прижати 2й прес
      AN    "y135";
      A     "y136";
      AN    "y134";
      AN    "y133";
      =     "y49";
NETWORK
TITLE = WE4.1 3 PRESS
//3 PRESS WORK SELECTED
//
      A(;
      A     #WorkSelect3Press;
      A     "x46";
      O;
      A     #WorkSelect3Press;
      A     "x47";
      O;
      A     #WorkSelect3Press;
      A     "x48";
      );
      A(;
      O     "y112";
      O     "y114";
      );
      S     "y150";
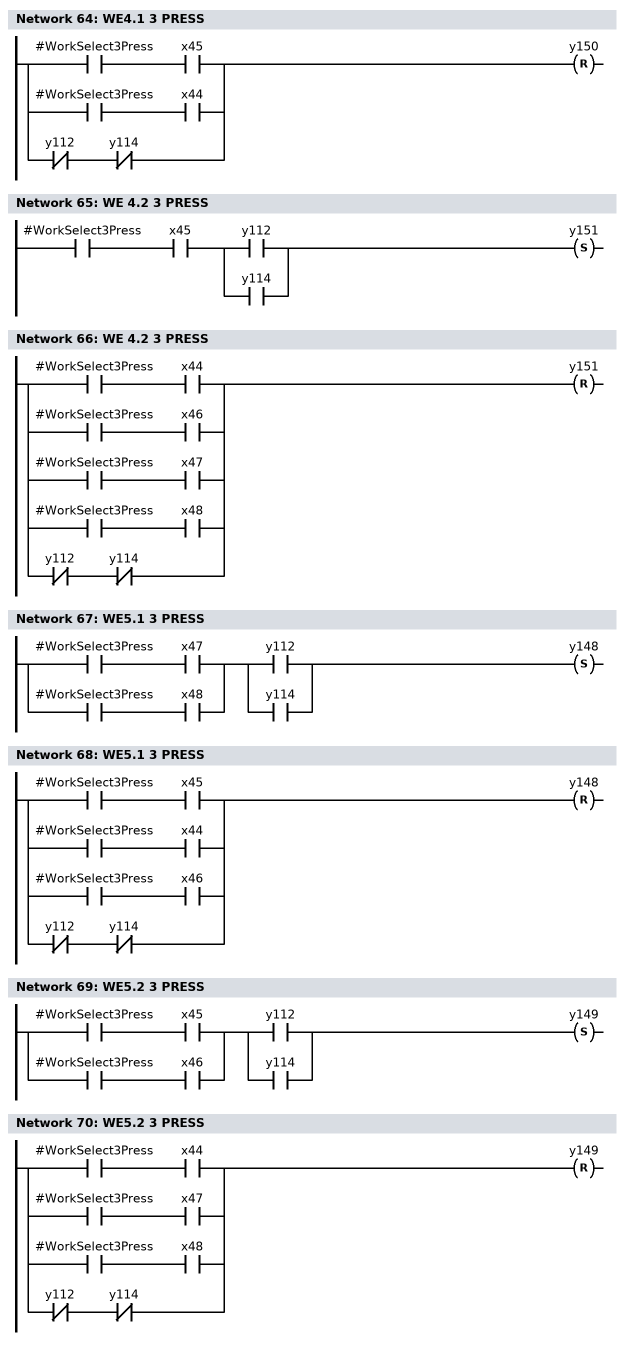
NETWORK
TITLE = WE4.1 3 PRESS
      A     #WorkSelect3Press;
      A     "x45";
      O;
      A     #WorkSelect3Press;
      A     "x44";
      O;
      AN    "y112";
      AN    "y114";
      R     "y150";
NETWORK
TITLE = WE 4.2 3 PRESS
      A     #WorkSelect3Press;
      A     "x45";
      A(;
      O     "y112";
      O     "y114";
      );
      S     "y151";
NETWORK
TITLE = WE 4.2 3 PRESS
      A     #WorkSelect3Press;
      A     "x44";
      O;
      A     #WorkSelect3Press;
      A     "x46";
      O;
      A     #WorkSelect3Press;
      A     "x47";
      O;
      A     #WorkSelect3Press;
      A     "x48";
      O;
      AN    "y112";
      AN    "y114";
      R     "y151";
NETWORK
TITLE = WE5.1 3 PRESS
      A(;
      A     #WorkSelect3Press;
      A     "x47";
      O;
      A     #WorkSelect3Press;
      A     "x48";
      );
      A(;
      O     "y112";
      O     "y114";
      );
      S     "y148";
NETWORK
TITLE = WE5.1 3 PRESS
      A     #WorkSelect3Press;
      A     "x45";
      O;
      A     #WorkSelect3Press;
      A     "x44";
      O;
      A     #WorkSelect3Press;
      A     "x46";
      O;
      AN    "y112";
      AN    "y114";
      R     "y148";
NETWORK
TITLE = WE5.2 3 PRESS
      A(;
      A     #WorkSelect3Press;
      A     "x45";
      O;
      A     #WorkSelect3Press;
      A     "x46";
      );
      A(;
      O     "y112";
      O     "y114";
      );
      S     "y149";
NETWORK
TITLE = WE5.2 3 PRESS
      A     #WorkSelect3Press;
      A     "x44";
      O;
      A     #WorkSelect3Press;
      A     "x47";
      O;
      A     #WorkSelect3Press;
      A     "x48";
      O;
      AN    "y112";
      AN    "y114";
      R     "y149";
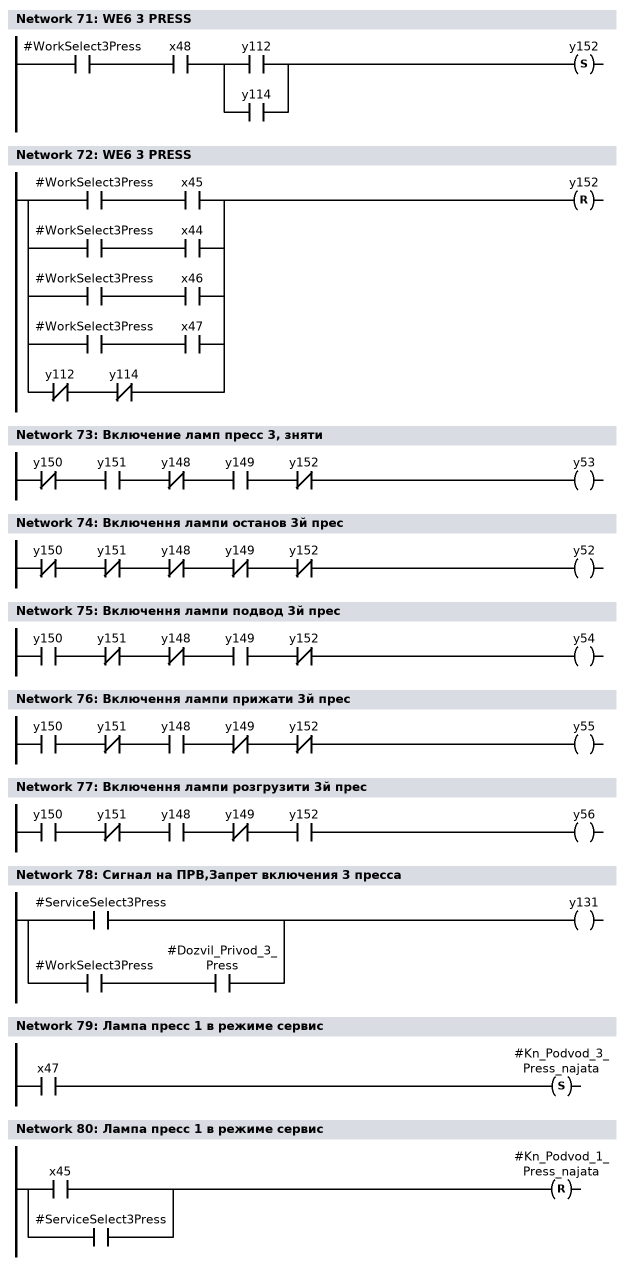
NETWORK
TITLE = WE6 3 PRESS
      A     #WorkSelect3Press;
      A     "x48";
      A(;
      O     "y112";
      O     "y114";
      );
      S     "y152";
NETWORK
TITLE = WE6 3 PRESS
      A     #WorkSelect3Press;
      A     "x45";
      O;
      A     #WorkSelect3Press;
      A     "x44";
      O;
      A     #WorkSelect3Press;
      A     "x46";
      O;
      A     #WorkSelect3Press;
      A     "x47";
      O;
      AN    "y112";
      AN    "y114";
      R     "y152";
NETWORK
TITLE = Включение ламп пресс 3, зняти 
      AN    "y150";
      A     "y151";
      AN    "y148";
      A     "y149";
      AN    "y152";
      =     "y53";
NETWORK
TITLE = Включення лампи останов 3й прес
      AN    "y150";
      AN    "y151";
      AN    "y148";
      AN    "y149";
      AN    "y152";
      =     "y52";
NETWORK
TITLE = Включення лампи подвод 3й прес
      A     "y150";
      AN    "y151";
      AN    "y148";
      A     "y149";
      AN    "y152";
      =     "y54";
NETWORK
TITLE = Включення лампи прижати 3й прес
      A     "y150";
      AN    "y151";
      A     "y148";
      AN    "y149";
      AN    "y152";
      =     "y55";
NETWORK
TITLE = Включення лампи розгрузити 3й прес
      A     "y150";
      AN    "y151";
      A     "y148";
      AN    "y149";
      A     "y152";
      =     "y56";
NETWORK
TITLE = Сигнал на ПРВ,Запрет включения 3 пресса
//Safery
//
      O     #ServiceSelect3Press;
      O;
      A     #WorkSelect3Press;
      A     #Dozvil_Privod_3_Press;
      =     "y131";
NETWORK
TITLE = Лампа пресс 1 в режиме сервис
      A     "x47";
      S     #Kn_Podvod_3_Press_najata;
NETWORK
TITLE = Лампа пресс 1 в режиме сервис
      O     "x45";
      O     #ServiceSelect3Press;
      R     #Kn_Podvod_1_Press_najata;
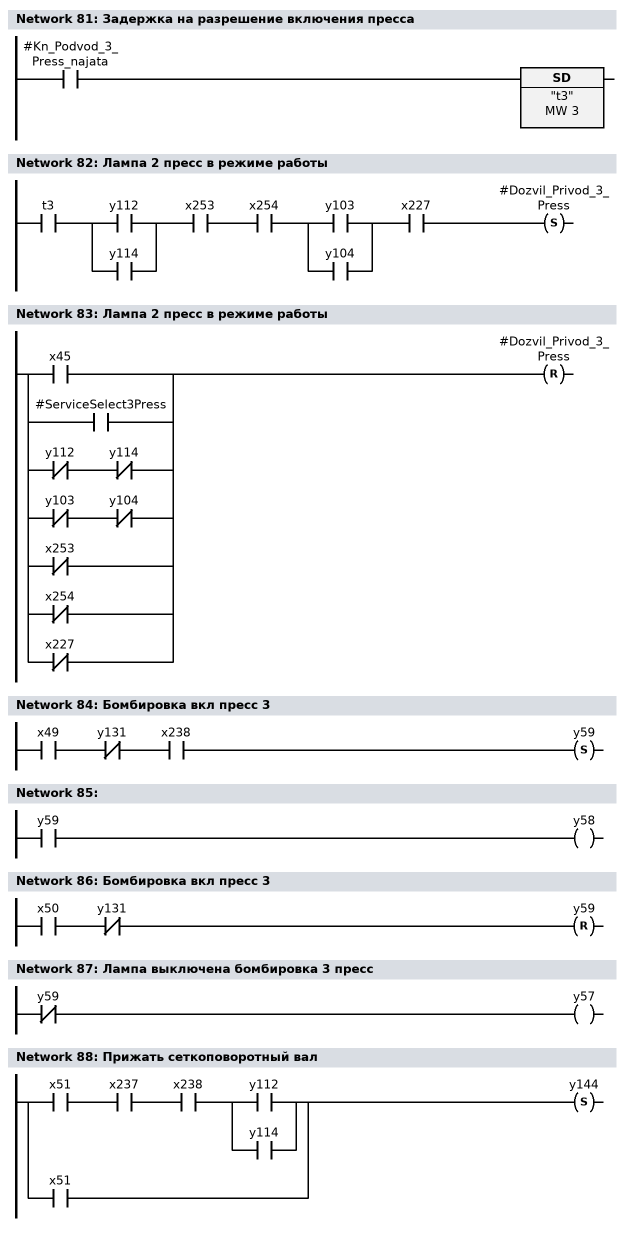
NETWORK
TITLE = Задержка на разрешение включения пресса
      A     #Kn_Podvod_3_Press_najata;
      L     MW 3;
      SD    "t3";
NETWORK
TITLE = Лампа 2 пресс в режиме работы
      A     "t3";
      A(;
      O     "y112";
      O     "y114";
      );
      A     "x253";
      A     "x254";
      A(;
      O     "y103";
      O     "y104";
      );
      A     "x227";
      S     #Dozvil_Privod_3_Press;
NETWORK
TITLE = Лампа 2 пресс в режиме работы
      O     "x45";
      O     #ServiceSelect3Press;
      O;
      AN    "y112";
      AN    "y114";
      O;
      AN    "y103";
      AN    "y104";
      ON    "x253";
      ON    "x254";
      ON    "x227";
      R     #Dozvil_Privod_3_Press;
NETWORK
TITLE = Бомбировка вкл пресс 3
      A     "x49";
      AN    "y131";
      A     "x238";
      S     "y59";
NETWORK
TITLE =
      A     "y59";
      =     "y58";
NETWORK
TITLE = Бомбировка вкл пресс 3
      A     "x50";
      AN    "y131";
      R     "y59";
NETWORK
TITLE = Лампа выключена бомбировка 3 пресс
      AN    "y59";
      =     "y57";
NETWORK
TITLE = Прижать сеткоповоротный вал
      A     "x51";
      A     "x237";
      A     "x238";
      A(;
      O     "y112";
      O     "y114";
      );
      O     "x51";
      S     "y144";
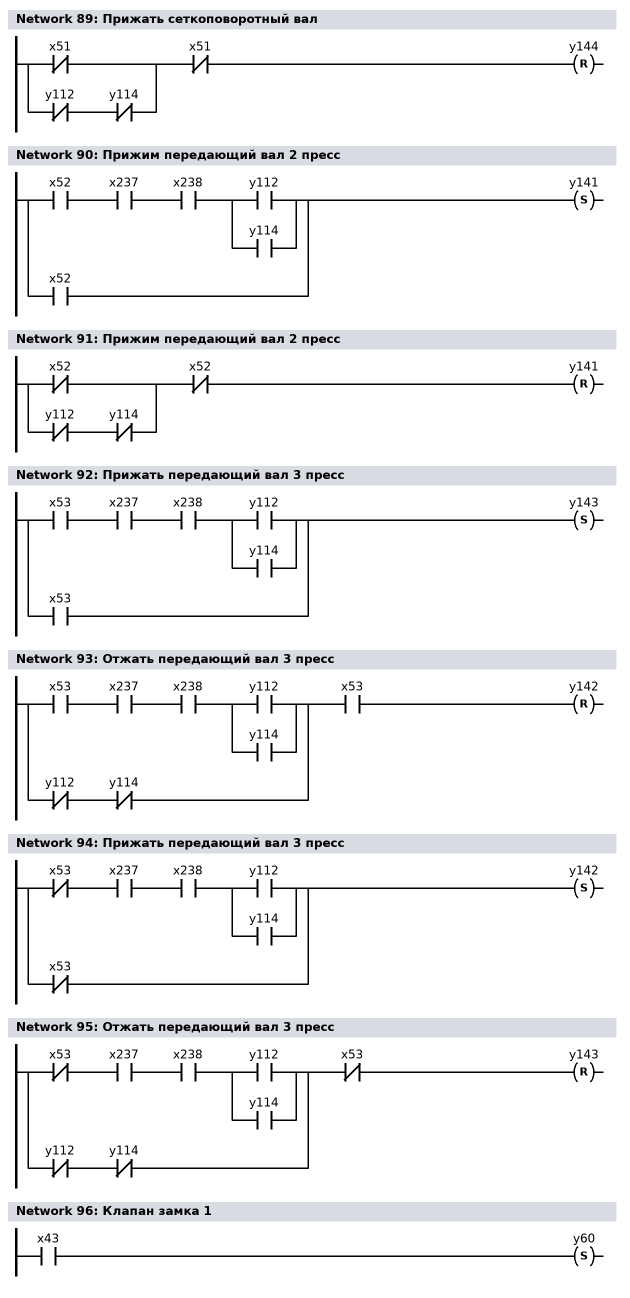
NETWORK
TITLE = Прижать сеткоповоротный вал
      A(;
      ON    "x51";
      O;
      AN    "y112";
      AN    "y114";
      );
      AN    "x51";
      R     "y144";
NETWORK
TITLE = Прижим передающий вал 2 пресс
      A     "x52";
      A     "x237";
      A     "x238";
      A(;
      O     "y112";
      O     "y114";
      );
      O     "x52";
      S     "y141";
NETWORK
TITLE = Прижим передающий вал 2 пресс
      A(;
      ON    "x52";
      O;
      AN    "y112";
      AN    "y114";
      );
      AN    "x52";
      R     "y141";
NETWORK
TITLE = Прижать передающий вал 3 пресс
      A     "x53";
      A     "x237";
      A     "x238";
      A(;
      O     "y112";
      O     "y114";
      );
      O     "x53";
      S     "y143";
NETWORK
TITLE = Отжать передающий вал 3 пресс
      A(;
      A     "x53";
      A     "x237";
      A     "x238";
      A(;
      O     "y112";
      O     "y114";
      );
      O;
      AN    "y112";
      AN    "y114";
      );
      A     "x53";
      R     "y142";
NETWORK
TITLE = Прижать передающий вал 3 пресс
      AN    "x53";
      A     "x237";
      A     "x238";
      A(;
      O     "y112";
      O     "y114";
      );
      ON    "x53";
      S     "y142";
NETWORK
TITLE = Отжать передающий вал 3 пресс
      A(;
      AN    "x53";
      A     "x237";
      A     "x238";
      A(;
      O     "y112";
      O     "y114";
      );
      O;
      AN    "y112";
      AN    "y114";
      );
      AN    "x53";
      R     "y143";
NETWORK
TITLE = Клапан замка 1
      A     "x43";
      S     "y60";
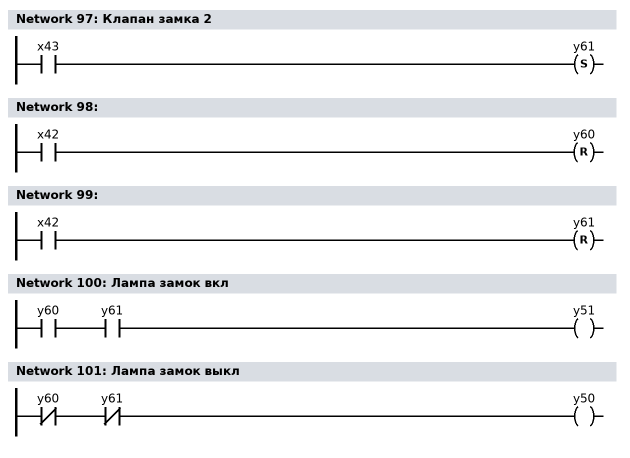
NETWORK
TITLE = Клапан замка 2
      A     "x43";
      S     "y61";
NETWORK
TITLE =
      A     "x42";
      R     "y60";
NETWORK
TITLE =
      A     "x42";
      R     "y61";
NETWORK
TITLE = Лампа замок вкл
      A     "y60";
      A     "y61";
      =     "y51";
NETWORK
TITLE = Лампа замок выкл
      AN    "y60";
      AN    "y61";
      =     "y50";
END_FUNCTION_BLOCK

DATA_BLOCK DB 11
VERSION : 0.0
"S-Walce"
BEGIN
END_DATA_BLOCK

DATA_BLOCK DB 12
VERSION : 0.0
"GS Bottom&Top Sprusk"
BEGIN
END_DATA_BLOCK

DATA_BLOCK DB 13
VERSION : 0.0
"Oscilation"
BEGIN
END_DATA_BLOCK

DATA_BLOCK DB 14
VERSION : 0.0
"Hihgt Preassure Clapan"
BEGIN
END_DATA_BLOCK

DATA_BLOCK DB 15
VERSION : 0.0
"Service&Work"
BEGIN
END_DATA_BLOCK

ORGANIZATION_BLOCK "CYCL_EXC"	// OB 1
TITLE = GydroA&B
VERSION : 0.1
VAR_TEMP
  OB1_EV_CLASS : BYTE ;	//Bits 0-3 = 1 (Coming event), Bits 4-7 = 1 (Event class 1)
  OB1_SCAN_1 : BYTE ;	//1 (Cold restart scan 1 of OB 1), 3 (Scan 2-n of OB 1)
  OB1_PRIORITY : BYTE ;	//Priority of OB Execution
  OB1_OB_NUMBR : BYTE ;	//1 (Organization block 1, OB1)
  OB1_RESERVED_1 : BYTE ;	//Reserved for system
  OB1_RESERVED_2 : BYTE ;	//Reserved for system
  OB1_PREV_CYCLE : INT ;	//Cycle time of previous OB1 scan (milliseconds)
  OB1_MIN_CYCLE : INT ;	//Minimum cycle time of OB1 (milliseconds)
  OB1_MAX_CYCLE : INT ;	//Maximum cycle time of OB1 (milliseconds)
  OB1_DATE_TIME : DATE_AND_TIME ;	//Date and time OB1 started
END_VAR
BEGIN
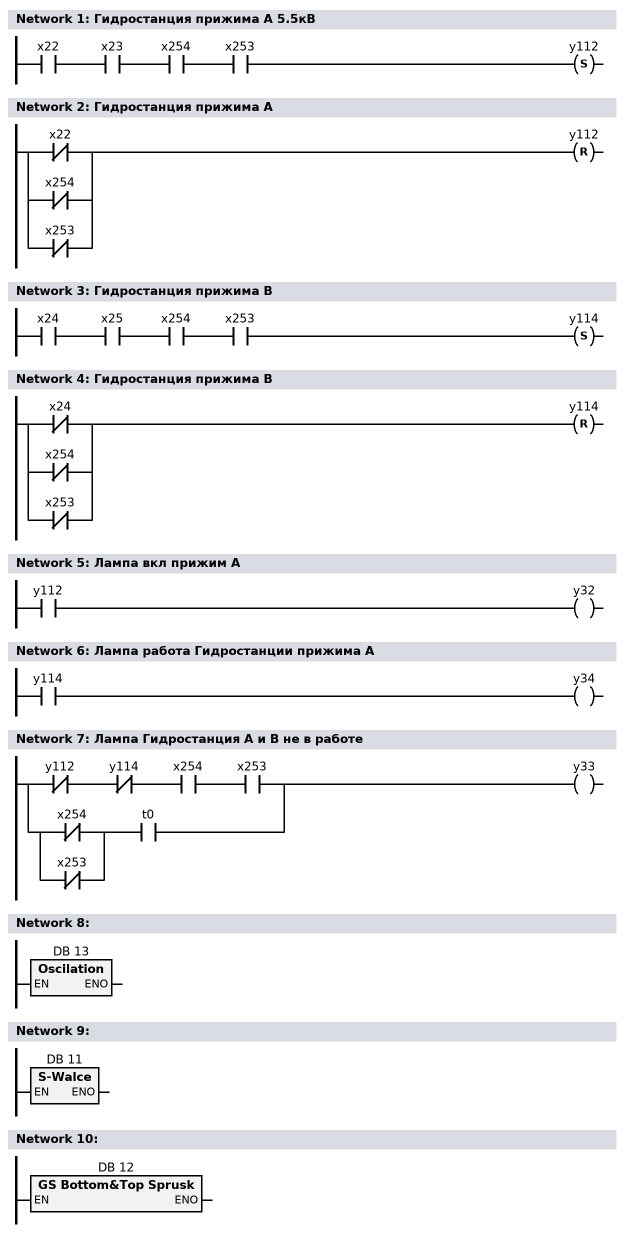
NETWORK
TITLE = Гидростанция прижима А 5.5кВ
      A     "x22";
      A     "x23";
      A     "x254";
      A     "x253";
      S     "y112";
NETWORK
TITLE = Гидростанция прижима А
      ON    "x22";
      ON    "x254";
      ON    "x253";
      R     "y112";
NETWORK
TITLE = Гидростанция прижима В
      A     "x24";
      A     "x25";
      A     "x254";
      A     "x253";
      S     "y114";
NETWORK
TITLE = Гидростанция прижима В
      ON    "x24";
      ON    "x254";
      ON    "x253";
      R     "y114";
NETWORK
TITLE = Лампа вкл прижим А
      A     "y112";
      =     "y32";
NETWORK
TITLE = Лампа работа Гидростанции прижима А
      A     "y114";
      =     "y34";
NETWORK
TITLE = Лампа Гидростанция А и В не в работе
      AN    "y112";
      AN    "y114";
      A     "x254";
      A     "x253";
      O;
      A(;
      ON    "x254";
      ON    "x253";
      );
      A     "t0";
      =     "y33";
NETWORK
TITLE =
      CALL  "Oscilation" , DB 13;
      NOP   0;
NETWORK
TITLE =
      CALL  "S-Walce" , DB 11;
      NOP   0;
NETWORK
TITLE =
      CALL  "GS Bottom&Top Sprusk" , DB 12;
      NOP   0;
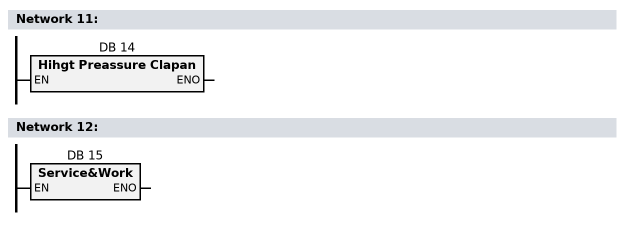
NETWORK
TITLE =
      CALL  "Hihgt Preassure Clapan" , DB 14;
      NOP   0;
NETWORK
TITLE =
      CALL  "Service&Work" , DB 15;
      NOP   0;
END_ORGANIZATION_BLOCK
